FUNCTION_BLOCK FB_Transfer
VAR_INPUT
	bExecute		: BOOL;
	stProcess		: REFERENCE TO ST_StageProcess;
	
	stSwing				: ST_CylinderInterface;
	fbSwing				: FB_Cylinder;
	stIncome			: ST_CylinderInterface;
	fbIncome			: FB_Cylinder;
	stIncomeCapture		: ST_CylinderInterface;
	fbIncomeCapture		: FB_Cylinder;
	stOutcome			: ST_CylinderInterface;
	fbOutcome			: FB_Cylinder;
	stOutcomeCapture	: ST_CylinderInterface;
	fbOutcomeCapture	: FB_Cylinder;
	
	bIncomeWorkOK		: BOOL;
	bOutcomeWorkOK		: BOOL;
END_VAR
VAR_OUTPUT
	bDone				: BOOL;
	bBusy				: BOOL;
	bActive				: BOOL;
	bError				: BOOL;
	sStateDiscrption	: WSTRING;
	wErrorID			: WORD;
END_VAR
VAR
	_step 					: INT := 0;
	_timer					: TON;
	_tSwingDelay			: TIME;
	_tIncomeDelay			: TIME;
	_tIncomeCaptureDelay	: TIME;
	_tOutcomedelay			: TIME;
	_tOutcomeCaptureDelay	: TIME;
END_VAR

CASE _step OF 
	0	: 
		sStateDiscrption := "State 0 : Init"; 	
		bDone := FALSE;
		bBusy := FALSE;
		bActive := FALSE;
		bError := FALSE;
		_timer(IN := FALSE);
		IF bActive THEN
			bBusy := TRUE;
			_step := 1;
		END_IF
	1	:
		sStateDiscrption := "State 1 : ";
		stSwing.bCmd := TRUE;
		IF 
END_CASE

END_FUNCTION_BLOCK

(* stored: Version 1.1.0.1, ProductVersion 3.1.4024.10
   POU FB_Transfer: Id {64a0402f-8352-4dbd-9e7d-b98eb4c48e03}, SpecialFunc None *)
